# EPICS substitutions: iocbio5/iocBoot/asynRecord.substitutions
file "$(ASYN)/db/asynRecord.db"
{
pattern
{P, R, PORT, ADDR, OMAX, IMAX}
{18ID:e:, asyn_1, ps1, 0, 256, 256}
}
